(* IEC 61131-3 sources: CodesysTest/export/Motion/PLCopen MC, 7 files *)

(* ---- MC_Halt.pou.st ---- *)
(*#-#-#-#-#-#-#-#-#-#---Declaration---#-#-#-#-#-#-#-#-#-#-#-#-#*)

FUNCTION_BLOCK FINAL MC_Halt EXTENDS MC_Base
VAR_INPUT
	Deceleration : REAL; 	// Value of the deceleration (decreasing energy of the motor) [u/s²]
END_VAR
VAR_OUTPUT
END_VAR
VAR
END_VAR
(*#-#-#-#-#-#-#-#-#-#---Implementation---#-#-#-#-#-#-#-#-#-#-#-#-#*)

//	Function Block: MC_Halt
//	Description: Commands a controlled motion stop. The axis is moved to the state DiscreteMotion, until the velocity is zero.
//				 When the output Done is set, the state is transferred to Standstill.
//	Created by: Ben Hess
//	Created Date: May 3rd, 2019

ExecuteOSR(CLK := Execute);

IF MC_State <> 0 AND Axis.Error THEN
	SetError();
	ErrorID := MC_ERROR.AXIS_ERROR_DURING_COMMAND;
	MC_State := 0;
	Axis.Halt := FALSE;
	Axis.AxisState := AXIS_STATE.AS_Standstill;
END_IF

CASE MC_State OF
	0:		// Idle State.  If execute rising edge then start halt
			IF ExecuteOSR.Q THEN
				IF NOT Axis.Error AND Axis.PowerState THEN
					SetBusy();
					Axis.AxisState := AXIS_STATE.AS_DiscreteMotion;
					Axis.QuickStopDeceleration := Deceleration;
					Axis.Halt := TRUE;
					MC_State := 1;
				ELSE
					Error := TRUE;
					ErrorID := MC_ERROR.AXIS_NOT_READY;
				END_IF

			END_IF

	1:		// Stopping.  Once stopped go back to idle
			IF Axis.ActVelocity = 0 THEN
				Axis.Halt := FALSE;
				Axis.AxisState := AXIS_STATE.AS_Standstill;
				SetDone();
				MC_State := 0;
			END_IF

	99: 		// Error
END_CASE

(* ---- MC_Home.pou.st ---- *)
(*#-#-#-#-#-#-#-#-#-#---Declaration---#-#-#-#-#-#-#-#-#-#-#-#-#*)

FUNCTION_BLOCK FINAL MC_Home EXTENDS MC_Base
VAR_INPUT
END_VAR
VAR_OUTPUT
END_VAR
VAR

END_VAR(*#-#-#-#-#-#-#-#-#-#---Implementation---#-#-#-#-#-#-#-#-#-#-#-#-#*)

//	Function Block: MC_Home
//	Description: Commands the axis to perform the «search home» sequence. The details of this sequence are manufacturer specific and can be set by the axis’ parameters.
//				 After completion, the axis state is Standstill if it was Standstill when started.
//	Created by: Ben Hess
//	Created Date: May 3rd, 2019

ExecuteOSR(CLK := Execute);

IF MC_State <> 0 AND Axis.Error THEN
	SetError();
	ErrorID := MC_ERROR.AXIS_ERROR_DURING_COMMAND;
	MC_State := 0;
	Axis.StartHoming := FALSE;
	Axis.AxisState := AXIS_STATE.AS_Standstill;
END_IF

CASE MC_State OF
	0:		// Idle State.  If execute rising edge then start halt
			IF ExecuteOSR.Q THEN
				IF NOT Axis.Error AND Axis.PowerState THEN
					SetBusy();
					Axis.AxisState := AXIS_STATE.AS_Homing;
					Axis.StartHoming := TRUE;
					MC_State := 1;
				ELSE
					Error := TRUE;
					ErrorID := MC_ERROR.AXIS_NOT_READY;
				END_IF
			END_IF

	1:		// Stopping.  Once stopped go back to idle
			IF Axis.HomingDone THEN
				Axis.StartHoming := FALSE;
				Axis.AxisState := AXIS_STATE.AS_Standstill;
				SetDone();
				MC_State := 0;
			ELSIF Axis.AxisState <> AXIS_STATE.AS_Homing THEN
				SetError();
				Axis.StartHoming := FALSE;
				MC_State := 0;
			END_IF
END_CASE

(* ---- MC_MoveAbsolute.pou.st ---- *)
(*#-#-#-#-#-#-#-#-#-#---Declaration---#-#-#-#-#-#-#-#-#-#-#-#-#*)

FUNCTION_BLOCK MC_MoveAbsolute EXTENDS MC_Base
VAR_INPUT
	Position : REAL;		// Commanded position for the motion (may be negative) (in technical units [u])
	Velocity : REAL;		// Value of the maximum velocity (always positive) (not necessarily reached) [u/s]
	Acceleration : REAL;	// Value of the acceleration (always positive) (increasing energy of the motor) [u/s²]
	Deceleration : REAL;	// Value of the deceleration (always positive) (decreasing energy of the motor) [u/s²]
END_VAR
VAR_OUTPUT
END_VAR
VAR
END_VAR
(*#-#-#-#-#-#-#-#-#-#---Implementation---#-#-#-#-#-#-#-#-#-#-#-#-#*)

//	Function Block: MC_MoveAbsolute
//	Description: Commands a controlled motion to a specified absolute position.
//				 After completion, the axis state is Standstill.
//	Created by: Ben Hess
//	Created Date: May 3rd, 2019

ExecuteOSR(CLK := Execute);
ExecuteOSF(CLK := Execute);

IF MC_State <> 0 AND Axis.Error THEN
	SetError();
	ErrorID := MC_ERROR.AXIS_ERROR_DURING_COMMAND;
	MC_State := 0;
	Axis.MoveAbs := FALSE;
END_IF

CASE MC_State OF
	0:		// Idle State.  If execute rising edge then start absolute move
			IF ExecuteOSR.Q THEN
				IF NOT Axis.Error AND Axis.PowerState THEN
					SetBusy();
					Axis.AxisState := AXIS_STATE.AS_DiscreteMotion;
					Axis.TargetPosDist := Position;
					Axis.ProfileVelocity := Velocity;
					Axis.ProfileAcceleration := Acceleration;
					Axis.ProfileDeceleration := Deceleration;
					Axis.ProfileCurrentLimit := Axis.DefaultCurrent;
					Axis.MoveAbs := TRUE;
					MC_State := 1;
					ErrorID := MC_ERROR.NO_ERROR;
				ELSE
					SetError();
					ErrorID := MC_ERROR.AXIS_NOT_READY;
				END_IF
			END_IF

	1:		// Wait for target reached.  Once stopped go back to idle
			IF Axis.TargetReached THEN
				Axis.MoveAbs := FALSE;
				SetDone();
				MC_State := 0;
			ELSIF Axis.AxisState <> AXIS_STATE.AS_DiscreteMotion OR CommandAborted THEN
				Axis.MoveAbs := FALSE;
				SetAborted();
				MC_State := 0;
			END_IF
END_CASE

(* ---- MC_MoveRelative.pou.st ---- *)
(*#-#-#-#-#-#-#-#-#-#---Declaration---#-#-#-#-#-#-#-#-#-#-#-#-#*)

FUNCTION_BLOCK MC_MoveRelative EXTENDS MC_Base
VAR_INPUT
	Distance : REAL;		// Relative distance for the motion (in technical units [u])
	Velocity : REAL;		// Value of the maximum velocity (always positive) (not necessarily reached) [u/s]
	Acceleration : REAL;	// Value of the acceleration (always positive) (increasing energy of the motor) [u/s²]
	Deceleration : REAL;	// Value of the deceleration (always positive) (decreasing energy of the motor) [u/s²]
END_VAR
VAR_OUTPUT
END_VAR
VAR
END_VAR
(*#-#-#-#-#-#-#-#-#-#---Implementation---#-#-#-#-#-#-#-#-#-#-#-#-#*)

//	Function Block: MC_MoveRelative
//	Description: Commands a controlled motion of a specified distance relative to the position at the time of the execution.
//				 The motion completes with velocity zero.
//				 After completion, the axis state is Standstill.
//	Created by: Ben Hess
//	Created Date: May 6th, 2019

ExecuteOSR(CLK := Execute);

IF MC_State <> 0 AND Axis.Error THEN
	SetError();
	ErrorID := MC_ERROR.AXIS_ERROR_DURING_COMMAND;
	MC_State := 0;
	Axis.MoveRel := FALSE;
	Axis.AxisState := AXIS_STATE.AS_ErrorStop;
END_IF

CASE MC_State OF
	0:		// Idle State.  If execute rising edge then start absolute move
			IF ExecuteOSR.Q THEN
				IF NOT Axis.Error AND Axis.PowerState THEN
					SetBusy();
					Axis.AxisState := AXIS_STATE.AS_DiscreteMotion;
					Axis.TargetPosDist := Distance;
					Axis.ProfileVelocity := Velocity;
					Axis.ProfileAcceleration := Acceleration;
					Axis.ProfileDeceleration := Deceleration;
					Axis.ProfileCurrentLimit := Axis.DefaultCurrent;
					Axis.MoveRel := TRUE;
					MC_State := 1;
					ErrorID := MC_ERROR.NO_ERROR;
				ELSE
					Error := TRUE;
					ErrorID := MC_ERROR.AXIS_NOT_READY;
				END_IF
			END_IF

	1:		// Wait for target reached.  Once stopped go back to idle
			IF Axis.TargetReached THEN
				Axis.MoveRel := FALSE;
				Axis.AxisState := AXIS_STATE.AS_Standstill;
				SetDone();
				MC_State := 0;
			ELSIF Axis.AxisState <> AXIS_STATE.AS_DiscreteMotion OR CommandAborted OR NOT Execute THEN
				Axis.MoveRel := FALSE;
				SetAborted();
				MC_State := 0;
			END_IF
END_CASE

(* ---- MC_Power.pou.st ---- *)
(*#-#-#-#-#-#-#-#-#-#---Declaration---#-#-#-#-#-#-#-#-#-#-#-#-#*)

FUNCTION_BLOCK MC_Power
VAR_INPUT
	Enable : BOOL; 			// Enables the FUNCTION block
	RegulatorOn : BOOL; 	// Enables the power stage
	DriveStart : BOOL; 		// Disables the quickstop mechanism
END_VAR
VAR_OUTPUT
	Status : BOOL; 					// Axis ready for motion
	RegulatorRealState : BOOL; 		// Effective state OF the power stage
	DriveStartRealState : BOOL; 	// Effective state of the quickstop mechanism
	Busy : BOOL; 					// Function block is executing
	Error : BOOL; 					// Signals that an error has occured
	ErrorID : MC_ERROR; 			// Error number
END_VAR
VAR
	EnableOSR : Standard.R_TRIG;
	MC_State : INT;
END_VAR
VAR_IN_OUT
	Axis : Axis_REF;		// Reference to the axis
END_VAR
(*#-#-#-#-#-#-#-#-#-#---Implementation---#-#-#-#-#-#-#-#-#-#-#-#-#*)

//	Function Block: MC_Power
//	Description: 	Controls the power stage of an axis and can be used to issue a quick stop.
//					◾A call of MC_Power_SML with bRegulatorOn=FALSE sets the axis state to PowerOff (disabled).
//					◾A call of MC_Power_SML with bRegulatorOn``=``TRUE on a disabled axis sets the axis state to Standstill, if there is no error on the axis. If an error is detected, the state of the axis is set to ErrorStop.
//					◾If the inputs Enable, bRegulatorOn and bDriveStart are ``TRUE but the output Status remains in FALSE for a long time, there may be a problem with the power stage, or an external halt may be set.
//					◾If power fails (also during operation), the axis state is set to ErrorStop.
//	Created by: Ben Hess
//	Created Date: May 6th, 2019

Status := Axis.PowerState AND Axis.EnableState;

RegulatorRealState := Axis.PowerState;
DriveStartRealState := Axis.EnableState;

IF NOT Enable THEN
	Axis.PowerOn := Axis.DriveEnable := FALSE;
ELSE
	Axis.PowerOn := RegulatorOn;
	Axis.DriveEnable := DriveStart;
END_IF

(* ---- MC_Reset.pou.st ---- *)
(*#-#-#-#-#-#-#-#-#-#---Declaration---#-#-#-#-#-#-#-#-#-#-#-#-#*)

FUNCTION_BLOCK FINAL MC_Reset EXTENDS MC_Base
VAR_INPUT
END_VAR
VAR_OUTPUT
END_VAR
VAR

END_VAR(*#-#-#-#-#-#-#-#-#-#---Implementation---#-#-#-#-#-#-#-#-#-#-#-#-#*)

//	Function Block: MC_Reset
//	Description: Forces the transition from the state ErrorStop to Standstill or PowerOff by resetting all internal axis-related errors.
//				 If the axis is not in state ErrorStop, the function block signals the error R_NO_ERROR_TO_RESET.
//	Created by: Ben Hess
//	Created Date: May 14th, 2019

ExecuteOSR(CLK := Execute);

IF MC_State <> 0 AND Axis.Error THEN
	SetError();
	ErrorID := MC_ERROR.AXIS_ERROR_DURING_COMMAND;
	MC_State := 0;
	Axis.AckError := FALSE;
END_IF

CASE MC_State OF
	0:		// Idle State.  If execute rising edge then start halt
			IF ExecuteOSR.Q THEN
				//IF Axis.Error THEN
					SetBusy();
					Axis.AckError := TRUE;
					MC_State := 1;
				//ELSE
				//	Error := TRUE;
				//	ErrorID := MC_ERROR.R_NO_ERROR_TO_RESET;
				//END_IF
			END_IF

	1:		// Clearing error.  Once stopped go back to idle
			IF NOT Axis.Error THEN
				Axis.AckError := FALSE;
				Axis.AxisState := AXIS_STATE.AS_Standstill;
				SetDone();
				MC_State := 0;
			END_IF
END_CASE

(* ---- MC_Stop.pou.st ---- *)
(*#-#-#-#-#-#-#-#-#-#---Declaration---#-#-#-#-#-#-#-#-#-#-#-#-#*)

FUNCTION_BLOCK FINAL MC_Stop EXTENDS MC_Base
VAR_INPUT
	Deceleration : REAL; 	// Value of the deceleration (decreasing energy of the motor) [u/s²]
END_VAR
VAR_OUTPUT
END_VAR
VAR
END_VAR
(*#-#-#-#-#-#-#-#-#-#---Implementation---#-#-#-#-#-#-#-#-#-#-#-#-#*)

//	Function Block: MC_Stop
//	Description: 	Executes a (blocking) stop on the axis.
//					As long as the Execute input is set or the stop is not finished, no other motion command is possible on the axis,
//					and the axis state is Stopping. After both the stop is finished and Execute is reset, the axis status is set to Standstill.

//	Created by: Ben Hess
//	Created Date: May 3rd, 2019

ExecuteOSR(CLK := Execute);

IF MC_State <> 0 AND Axis.Error THEN
	SetError();
	ErrorID := MC_ERROR.AXIS_ERROR_DURING_COMMAND;
	MC_State := 0;
	Axis.Halt := FALSE;
	Axis.AxisState := AXIS_STATE.AS_Standstill;
END_IF

CASE MC_State OF
	0:		// Idle State.  If execute rising edge then start halt
			IF ExecuteOSR.Q THEN
				IF NOT Axis.Error AND Axis.PowerState THEN
					SetBusy();
					Axis.AxisState := AXIS_STATE.AS_DiscreteMotion;
					Axis.QuickStopDeceleration := Deceleration;
					Axis.Halt := TRUE;
					MC_State := 1;
				ELSE
					Error := TRUE;
					ErrorID := MC_ERROR.AXIS_NOT_READY;
				END_IF

			END_IF

	1:		// Stopping.  Once stopped go back to idle
			IF Axis.ActVelocity = 0 THEN
				Axis.Halt := FALSE;
				Axis.AxisState := AXIS_STATE.AS_Standstill;
				SetDone();
				MC_State := 0;
			END_IF

	99: 		// Error
END_CASE
